// TIA Portal V20 export
TYPE "LKinCtrl_Utilities_typeNewTableConfiguration"
// stored: Access Published
   STRUCT
      lowerBoundArray { ExternalAccessible := 'False'; ExternalVisible := 'False'; ExternalWritable := 'False'} : DInt;   // Lower bound of the array to be displayed in the table window.
      upperBoundArray { ExternalAccessible := 'False'; ExternalVisible := 'False'; ExternalWritable := 'False'} : DInt;   // Upper bound of the array to be displayed in the table window.
      emptyTable { ExternalAccessible := 'False'; ExternalVisible := 'False'; ExternalWritable := 'False'} : Bool;   // TRUE: The table is empty. No selection, no interactivity.
      sizeTableWindow { ExternalAccessible := 'False'; ExternalVisible := 'False'; ExternalWritable := 'False'} : Int := 1;   // Number of elements that can be displayed at once in the table window.
      fieldsToSkip { ExternalAccessible := 'False'; ExternalVisible := 'False'; ExternalWritable := 'False'} : Int := 1;   // Number of fields to skip when button up or down is pressed.
   END_STRUCT;
END_TYPE
